# EPICS autosave request: ADADSC/iocs/adscIOC/iocBoot/iocAdsc/auto_settings.req
file "adsc_settings.req", P=$(P), R=det1:
